# EPICS autosave request: iocBoot/generic_motors_ioc/dbSave/bluiceRuns.req
$(P)runCount
$(P)currentRun
$(P)isActive
$(P)doseMode
$(P)updated
$(P)currentUser
